// TwinCAT 3 PLC project PLC3
// ProgramVersion: 3.1.4023.0
// libraries:
//   Tc2_Standard, * (Beckhoff Automation GmbH)
//   Tc2_System, * (Beckhoff Automation GmbH)
//   Tc3_Module, * (Beckhoff Automation GmbH)
// project tree:
//   / PlcTask.TcTTO (not stored)
//   POUs/ FB_Base.TcPOU (not stored), FB_Child.TcPOU, I_Interface2.TcIO (not stored), I_Interface.TcIO (not stored), MAIN.TcPOU (not stored)
// real-time tasks:
//   TASK PlcTask: cycle T#10ms, priority 20, ADS port 350

// ---- POUs/FB_Child.TcPOU
FUNCTION_BLOCK  FB_Child EXTENDS FB_Base  IMPLEMENTS I_Interface,I_Interface2

VAR_INPUT
END_VAR
VAR
    
SomeText: STRING;
	Counter		: DINT:= 1 ;
  Result		: DINT :=2;
    
    
      Base:FB_Base;
END_VAR

SomeText:= 'Current counts';

IF Conditions[1] AND Conditions[2]  AND Conditions[3] AND Conditions[4] AND Conditions[5]AND Conditions[6] THEN
	Counter :=Counter+ 1;

	IF Counter > 2 THEN
	Counter := Counter + 5 ;
	END_IF
END_IF

Base(Variable1:=2, Variable2:=3 , Variable3:= 5,Sentence:='', Conditions :=Conditions);


AddTwoInts(    Variable1 :=4,
    Variable2:=4);

METHOD AddTwoInts:DINT
VAR_INPUT
  Variable1 :DINT;
    Variable2:DINT ;
END_VAR
AddTwoInts:=Variable1+Variable2 ;
END_METHOD

END_FUNCTION_BLOCK
